PROGRAM TestingEvents
VAR
	bIsInitalized : BOOL;
    fbMessage : FB_TcMessage;
    bSendMessage : BOOL;
	
	bIsAlarmInit : BOOL;
	fbAlarm : FB_TcAlarm;
	bRaiseAlarm : BOOL;
	bClearAlarm : BOOL;
	bConfirmAlarm : BOOL;
END_VAR

IF NOT bIsInitalized THEN
    bIsInitalized := TRUE;
    fbMessage.CreateEx(TC_Events.MyEvents.Start, 0);
END_IF

IF bSendMessage THEN
    bSendMessage := FALSE;
    fbMessage.Send(0); //Current timestamp
END_IF

IF NOT bIsAlarmInit THEN
	bIsAlarmInit := TRUE;
	fbAlarm.CreateEx(TC_Events.MyEvents.Stop, TRUE, 0);
END_IF

IF bRaiseAlarm THEN
	bRaiseAlarm := FALSE;
	fbAlarm.ipArguments.Clear().AddString('The axis that is running');
	fbAlarm.Raise(0);
END_IF

IF bConfirmAlarm THEN
    bConfirmAlarm := FALSE;
    fbAlarm.Confirm(0);
END_IF

IF bClearAlarm THEN
    bClearAlarm := FALSE;
    fbAlarm.Clear(0, FALSE);
END_IF

END_PROGRAM

(* stored: Version 1.1.0.1, ProductVersion 3.1.4024.11
   POU TestingEvents: Id {a26af1e2-89c2-42bc-b830-9454228f9dcd}, SpecialFunc None *)
